{attribute addProperty BoxType "AX8108-0000-0041-0041"}
{attribute addProperty Id "Power_supply_statuswordAT %Q*UINT162"}
{attribute addProperty CRC "69469960"}
{attribute addProperty SizeInBites "16"}
{attribute addProperty SizeInBytes "2"}
TYPE DeviceMain_Outputs_04240708 :
STRUCT
	{attribute addProperty Name "Power_supply_statusword"}
	Power_supply_statusword AT %Q* : UINT;
END_STRUCT
END_TYPE

(* stored: Version 1.2.0.0, ProductVersion 3.1.4024.9
   DUT DeviceMain_Outputs_04240708: Id {8358d2ce-33e3-4557-82cf-9bec49518c3a} *)
